FUNCTION IsRoiSizeOK : BOOL
VAR_INPUT
    RoiRectangle : TcVnRectangle_UDINT;
    ImageWidth : UDINT;
    ImageHeight : UDINT;
END_VAR

IF NOT (RoiRectangle.nX < ImageWidth) THEN
	RETURN;
END_IF

IF NOT (RoiRectangle.nY < ImageHeight) THEN
	RETURN;
END_IF

IF NOT (RoiRectangle.nWidth <= (ImageWidth - RoiRectangle.nX)) THEN
	RETURN;
END_IF

IF NOT (RoiRectangle.nHeight <= (ImageHeight - RoiRectangle.nY)) THEN
	RETURN;
END_IF

IsRoiSizeOK := TRUE;

END_FUNCTION

(* stored: Version 1.1.0.1, ProductVersion 3.1.4024.13
   POU IsRoiSizeOK: Id {b638c6eb-8eba-0128-1111-5151f88af721}, SpecialFunc None *)
